# EPICS substitutions: examples/ExampleApp/Db/user.substitutions
# Example substitutions file

file "db/circle.db" {
    { user = "training" }
}

file "db/dbExample1.db" {
    { user = "training" }
}

file db/dbExample2.db {
    pattern { user, no, scan }
        { "training", 1, "1 second" }
        { "training", 2, "2 second" }
        { "training", 3, "5 second" }
}
